DATA_BLOCK "10_PN_NETWORK"
{ DB_Accessible_From_OPC_UA := 'FALSE' ;
 DB_Accessible_From_Webserver := 'FALSE' ;
 S7_Optimized_Access := 'TRUE' }
VERSION : 0.1
NON_RETAIN
   VAR
      SUBNET_10 : Array[0..1023] of Bool;   // one array per subnet
   END_VAR


BEGIN

END_DATA_BLOCK

